INTERFACE I_MotionInterlock


METHOD CanMoveNegative : BOOL
END_METHOD


METHOD CanMovePositive : BOOL
END_METHOD


METHOD CanPowerOn : BOOL
END_METHOD

END_INTERFACE

(* stored: Version 1.1.0.1
   Itf I_MotionInterlock: Id {72cf8f13-457a-43cf-915b-628c96ed4ea0}
   Method CanMoveNegative: Id {b07a61a3-1e40-445e-a098-36ca243a9ed4}
   Method CanMovePositive: Id {6adf3334-0372-45b3-8a70-e9dca85dbba7}
   Method CanPowerOn: Id {019d2a14-8f32-4838-a078-8b1e90eb609f} *)
